(* IEC 61131-3 sources: AXOpen/src/integrations/app/src/Examples/AXOpen.AxoObject, 1 file *)

(* ---- AxoObjectExample.st ---- *)
USING AXOpen.Core;

NAMESPACE AxoObjectExamples
//<AxoContext>
    {S7.extern=ReadWrite}
    CLASS PUBLIC MyContext EXTENDS  AXOpen.Core.AxoContext
        VAR
            _myObject : AxoObject;
        END_VAR
        METHOD PROTECTED OVERRIDE Main
            _myObject.InitializeWithContext(THIS);
        END_METHOD
    END_CLASS
//</AxoContext>
//<AxoObject>
    {S7.extern=ReadWrite}
    CLASS PUBLIC MyParentObject  EXTENDS AxoContext
        VAR
            _myChildObject  : AxoObject;
        END_VAR
        METHOD PROTECTED OVERRIDE Main
            _myChildObject.InitializeWithContext(THIS);
        END_METHOD
    END_CLASS
//</AxoObject>
END_NAMESPACE
